// TIA Portal V18 export
// export: Created 2025-12-01T17:53:16.0252984Z, ExportSetting None, DisplayName Totally Integrated Automation Portal, DisplayVersion V18 Update 5, DisplayName TIA Portal Openness, DisplayVersion V18 Update 5, DisplayName TIA Portal Teamcenter Gateway, DisplayVersion V18, DisplayName TIA Portal Version Control Interface, DisplayVersion V18, DisplayName STEP 7 Professional, DisplayVersion V18 Update 5, DisplayName STEP 7 Safety, DisplayVersion V18, DisplayName WinCC Professional, DisplayVersion V18 Update 5
Screen "490PDF Manual"  1280x800, Number=490, Template=04Information
  ScreenLayer 
    Button "按钮_1"  StyleItem=BtnFunction20, TextOff="缩小 / Zoom Out / Oddialiť"
      on Click: PDFZoomOut(Screen object := PDFView_1)
    Button "按钮_2"  StyleItem=BtnFunction20, TextOff="放大 / Zoom In / Priblížiť"
      on Click: PDFZoomIn(Screen object := PDFView_1)
    Button "按钮_3" at 1152,350 size 128x75  StyleItem=BtnFunction20, TextOff="向下 / Down / Dole"
      on Click: PDFScrollDown(Screen object := PDFView_1)
    Button "btnMenu8_1"  StyleItem=BtnFunction20, TextOff="右移 / Scroll Right / Posuňte sa doprava"
      on Click: PDFScrollRight(Screen object := PDFView_1)
    Button "btnMenu8_2"  StyleItem=BtnFunction20, TextOff="自适应 / Auto Adaption / Auto Adaptácia"
      on Click: PDFFitToHeight(Screen object := PDFView_1); PDFFitToWidth(Screen object := PDFView_1)
    Button "按钮_4" at 1152,435 size 128x75  StyleItem=BtnFunction20, TextOff="下一页 / Next / Budúci"
      on Click: PDFGotoNextPage(Screen object := PDFView_1)
    Button "按钮_5" at 1152,520 size 128x75  StyleItem=BtnFunction20, TextOff="末页 / End / Koniec"
      on Click: PDFGotoLastPage(Screen object := PDFView_1)
    Button "按钮_6" at 1152,180 size 128x75  StyleItem=BtnFunction20, TextOff="前一页 / Previous / Predchádzajúci"
      on Click: PDFGotoPreviousPage(Screen object := PDFView_1)
    Button "btnMenu8_3"  StyleItem=BtnFunction20, TextOff="左移 / Scroll Left / Posuňte sa doľava"
      on Click: PDFScrollLeft(Screen object := PDFView_1)
    Button "btnMenu8_4"  StyleItem=BtnFunction20, TextOff="选择 PDF文件 / Select PDF file / Vybrať Súbor PDF"
      on Click: OpenFileBrowser(Mask := *.pdf*, Start folder := C:, File := 1, Navigation back := 1, Navigation up := 1, New folder := 0, Path := BrowseFile, Status := BrowseStatus)
    Button "按钮_7" at 1152,95 size 128x75  StyleItem=BtnFunction20, TextOff="首页 / Home / Domov"
      on Click: PDFGotoFirstPage(Screen object := PDFView_1)
    Button "按钮_8" at 1152,265 size 128x75  StyleItem=BtnFunction20, TextOff="向上 / UP / HORE"
      on Click: PDFScrollUp(Screen object := PDFView_1)
    Group "Group"
      TextField "Text field_1"  StyleItem=Textfeld, Text="路径: / Path： / Cestička:"
      IOField "I/O field_1"  DataFormat=String, FormatPattern=????????????????????????????????????????????????????????????????????????????????, Mode=Output, StyleItem=IO Input22
        ProcessValue := BrowseFile
    Button "btnMenu8_5" at 1152,605 size 128x75  StyleItem=BtnFunction18
    Button "btnMenu8_7"  StyleItem=BtnFunction18
    Button "btnMenu7" at 1018,724 size 128x75  StyleItem=BtnActive20, TextOff="PDF 手册 / PDF Manual / PDF Manuálny"
      on Click: ActivateScreen(Screen name := , Object number := 0); SetTag(Tag := Sys_VersionManagement_HMIPageID, Value := 490)
